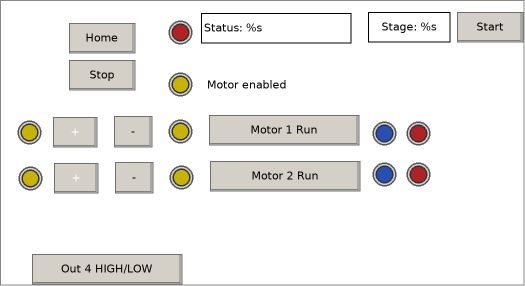
VISUALIZATION HMI1  // 525x286
    Button (53,117 44x30), "+"
        OnMouseClick: execute {
            MAINVARS.BitOut0 := FALSE;
            MAINVARS.BitOut1 := TRUE;
            MAINVARS.BitOut2 := TRUE;
        }
        OnMouseLeave: execute { MAINVARS.BitOut0 := TRUE; }
    Button (114,116 38x31), "-"
        OnMouseClick: execute {
            MAINVARS.BitOut0 := FALSE;
            MAINVARS.BitOut1 := FALSE;
            MAINVARS.BitOut2 := TRUE;
        }
        OnMouseLeave: execute { MAINVARS.BitOut0 := TRUE; }
    Button (69,23 66x30), "Home"
    Lamp1 (16,119 27x27), variable: MAINVARS.BitOut1 = TRUE;, style: Lamp-Lamp1-Yellow
    Lamp1 (167,71 27x27), variable: MAINVARS.BitOut0 = FALSE OR MAINVARS.BitOut5 = FALSE;, style: Lamp-Lamp1-Yellow
    Label (204,70 94x30), "Motor enabled"
    Lamp1 (167,118 27x27), variable: MAINVARS.BitOut1 = FALSE;, style: Lamp-Lamp1-Yellow
    Lamp1 (167,19 27x27), variable: MAINVARS.GlobalAlarm, style: Lamp-Lamp1-Red
    Rectangle (201,13 150x30), "Status: %s", text variable: MAINVARS.AlarmMessage
    Button (69,60 66x30), "Stop"
        OnMouseClick: execute {
            MAINVARS.BitOut0 := TRUE;
            MAINVARS.BitOut2 := FALSE;
            MAINVARS.Start := FALSE;
            MAINVARS.AlarmMessage := 'Stopped';
            MAINVARS.MachineState := 0;
            MAINVARS.PreviousMachineState := 0;
        }
    Rectangle (368,12 82x30), "Stage: %s", text variable: MAINVARS.MachineState
    Button (457,12 66x30), "Start"
        OnMouseClick: toggle MAINVARS.Start
    Button (209,115 150x30), "Motor 1 Run"
        OnMouseClick: execute { MAINVARS.BitOut2 := TRUE; }
        OnMouseUp: execute { MAINVARS.BitOut2 := FALSE; }
    Button (32,254 150x30), "Out 4 HIGH/LOW"
        toggle MAINVARS.BitOut3
    Button (54,163 44x30), "+"
        OnMouseClick: execute {
            MAINVARS.BitOut5 := FALSE;
            MAINVARS.BitOut6 := TRUE;
            MAINVARS.BitOut7 := TRUE;
        }
        OnMouseLeave: execute { MAINVARS.BitOut5 := TRUE; }
    Button (115,162 38x31), "-"
        OnMouseClick: execute {
            MAINVARS.BitOut5 := FALSE;
            MAINVARS.BitOut6 := FALSE;
            MAINVARS.BitOut7 := TRUE;
        }
        OnMouseLeave: execute { MAINVARS.BitOut5 := TRUE; }
    Lamp1 (17,165 27x27), variable: MAINVARS.BitOut6 = TRUE;, style: Lamp-Lamp1-Yellow
    Lamp1 (168,164 27x27), variable: MAINVARS.BitOut6 = FALSE;, style: Lamp-Lamp1-Yellow
    Button (210,161 150x30), "Motor 2 Run"
        OnMouseClick: execute { MAINVARS.BitOut2 := TRUE; }
        OnMouseUp: execute { MAINVARS.BitOut2 := FALSE; }
    Lamp1 (371,120 27x27), variable: MAINVARS.BitIn4 = FALSE, style: Lamp-Lamp1-Blue
    Lamp1 (371,161 27x27), variable: MAINVARS.BitIn5 = FALSE, style: Lamp-Lamp1-Blue
    Lamp1 (405,120 27x27), variable: MAINVARS.BitIn0 = FALSE, style: Lamp-Lamp1-Red
    Lamp1 (405,161 27x27), variable: MAINVARS.BitIn2 = FALSE, style: Lamp-Lamp1-Red
END_VISUALIZATION

(* stored: Version 1.1.0.1, ProductVersion 3.1.4024.2
   Visu HMI1: Id {22e1470a-977b-4397-b4ed-ebfb4665ff6a} *)
